Fanuc KAREL source: ko00077.KL

-- PROVISIONAL review KL for V1013-1; original PC SHA256 ac21982b7750a7a74bfd8c18bed47da3a6e2bad4d0aeb46b54208b6c0d39e76b
-- Incomplete behavior may be omitted. Consult companion uncertainty JSON. Do not deploy.
PROGRAM KO00077
%NOLOCKGROUP
BEGIN
  -- UNRESOLVED_PC offsets 5-12; opcodes 9D,23
  -- UNRESOLVED_PC offsets 17-66; opcodes 27,22,1C,27,49,7E,AD,22,31,7E,4A
  -- UNRESOLVED_PC offsets 71-75; opcodes 7F
END KO00077
